INTERFACE IPathQuery3

METHOD ReserveAsync
VAR_INPUT
  unit : REFERENCE TO Unit;
END_VAR
END_METHOD

END_INTERFACE

(* stored: Version 1.1.0.1
   Itf IPathQuery3: Id {4a888ebc-659c-45c3-a9f4-41422609cae5}
   Method ReserveAsync: Id {b4ac4429-c892-41f9-a83b-a581dc75caad} *)
